// TIA Portal project "Robin_automation" (V16)
// Vorlageprojekt für das Buch mit Zielsystem S7-1200

(* hardware
DEVICE "S7-1200-Station_1"  S7-1200 Station
   slot 0: "Baugruppenträger_0"  Rack  V1.0
   slot 1: "PLC_1"  CPU 1211C DC/DC/DC  6ES7 211-1AE40-0XB0  V4.1
*)

// ===== PLC "PLC_1"  CPU 1211C DC/DC/DC =====

VAR_GLOBAL   // PLC tag table "Standard-Variablentabelle"
   "Start Button 1" AT %I0.0 : Bool;
   "Stop Button 1" AT %I0.1 : Bool;
   "Emergency Stop 1" AT %I0.2 : Bool;
   "Roller Conveyor (2m) 2" AT %Q0.0 : Bool;
   "Belt Conveyor (4m) 3" AT %Q0.1 : Bool;
   "Diffuse Sensor 1" AT %I0.3 : Bool;
   "Loadong Conveyor 1" AT %Q0.2 : Bool;
   "Diffuse Sensor 4" AT %I0.4 : Bool;
   "Diffuse Sensor 2" AT %I0.5 : Bool;
   "Chain Transfer 3 (+)" AT %Q0.4 : Bool;
   "Chain Transfer 3 (Right)" AT %Q0.5 : Bool;
   "Chain Transfer 3 (Left)" AT %Q0.6 : Bool;
   "Chain Transfer 1 (Left)" AT %Q0.7 : Bool;
   "Chain Transfer 1 (+)" AT %Q1.0 : Bool;
   "Chain Transfer 2 (Right)" AT %Q1.1 : Bool;
   "Chain Transfer 2 (+)" AT %Q1.2 : Bool;
   "Belt Conveyor (4m) 2" AT %Q1.3 : Bool;
   "Belt Conveyor (4m) 1" AT %Q1.4 : Bool;
   "Diffuse Sensor 6" AT %I0.6 : Bool;
   "Diffuse Sensor 3" AT %I0.7 : Bool;
   "Diffuse Sensor 7" AT %I1.0 : Bool;
   "Diffuse Sensor 8" AT %I1.1 : Bool;
   "Tag_1" AT %M0.0 : Bool;
   "Tag_2" AT %M0.1 : Bool;
   "Stack Light 1 (Green)" AT %Q1.7 : Bool;
   "Stack Light 1 (Yellow)" AT %Q1.6 : Bool;
   "Tag_3" AT %M0.3 : Bool;
   "Barkod Bitti" AT %I1.2 : Bool;
   "Loading Conveyor 2" AT %Q1.5 : Bool;
   "Tag_4" AT %M0.5 : Bool;
   "Tag_5" AT %M0.4 : Bool;
   "Tag_6" AT %M1.0 : Bool;
   "Tag_7" AT %M2.0 : Bool;
   "Diffuse Sensor 5" AT %I1.3 : Bool;
   "Tag_8" AT %M2.1 : Bool;
   "Tag_9" AT %M3.0 : Bool;
   "Start Button 3" AT %I1.4 : Bool;
   "Tag_10" AT %M3.1 : Bool;
   "Tag_11" AT %M1.1 : Bool;
   "Tag_12" AT %M1.2 : Bool;
   "Tag_13" AT %M1.3 : Bool;
   "Tag_14" AT %M0.2 : Bool;
   "Tag_15" AT %M1.4 : Bool;
   "Tag_16" AT %M1.5 : Bool;
   "Tag_17" AT %M1.6 : Bool;
   "Tag_18" AT %M1.7 : Bool;
   "Tag_19" AT %M0.6 : Bool;
   "Sağ boş  Sol dolu ise AÇIK" AT %M0.7 : Bool;
   "Tag_20" AT %M2.2 : Bool;
   "Tag_21" AT %M2.3 : Bool;
   "Tag_22" AT %M2.5 : Bool;
   "Tag_23" AT %M2.6 : Bool;
   "Tag_24" AT %M2.7 : Bool;
END_VAR

TYPE "User_data_type_1"
   STRUCT
      "Start Button" : Bool;
   END_STRUCT;
END_TYPE

FUNCTION "MHJ-PLC-Lab-Function-S71200" : Void   // FC9000, SCL
{ S7_Optimized_Access := 'TRUE' }
VERSION : 0.1
   VAR_TEMP
      rdTimeReturn : Int;
      outputTime : DTL;
      SyncVal : Byte;
      forVal : Int;
      forVal_2 : Int;
      Value : Byte;
   END_VAR
   VAR CONSTANT
      CompVal : Byte := 16#34;
      Value_01 : Byte := 16#11;
      Value_01_DW : DWord := 16#A165_D992;
      Value_02_DW : DWord := 16#58BE_4401;
   END_VAR
BEGIN

   #Value:=PEEK(area := 16#82,
        dbNumber := 0,
        byteOffset := 511);
   #Value := #Value + 1;

   POKE(area := 16#82,
        dbNumber := 0,
        byteOffset := 511,
        value := #Value);

   POKE(area:=16#81,
        dbNumber:=0,
        byteOffset:=1016,
        value:=#Value_01_DW);
   POKE(area := 16#81,
        dbNumber := 0,
        byteOffset := 1020,
        value := #Value_02_DW);

   POKE(area := 16#81,
        dbNumber := 0,
        byteOffset := 511,
        value := B#16#00);

   FOR #forVal := 0 TO 120 DO
       FOR #forVal_2:=0 TO 10 DO
           #rdTimeReturn:=RD_SYS_T(#outputTime);
           #rdTimeReturn := WR_SYS_T(#outputTime);
           #rdTimeReturn := RD_SYS_T(#outputTime);
           #rdTimeReturn := WR_SYS_T(#outputTime);
       END_FOR;
       #SyncVal:= PEEK(area := 16#81,
                      dbNumber := 0,
                      byteOffset := 511);
       IF #SyncVal = #CompVal THEN
          GOTO M_1;
       END_IF;
   END_FOR;
   RETURN;

   M_1:
   POKE(area := 16#81,
        dbNumber := 0,
        byteOffset := 511,
        value := B#16#0);
END_FUNCTION

// folder: System blocks/Program resources

ORGANIZATION_BLOCK "Main"   // OB1, LAD, ProgramCycle
TITLE = "Main Program Sweep (Cycle)"
{ S7_Optimized_Access := 'TRUE' }
VERSION : 0.1
   VAR_INPUT
      Initial_Call : Bool;   // Initial call of this OB
      Remanence : Bool;   // =True, if remanent data are available
   END_VAR
   VAR_TEMP   // added for the SCL form of the ladder/FBD networks
      _w1 : Bool;
      _w2 : Bool;
   END_VAR
BEGIN

REGION Network 1: Konnektierungsbaustein für PLC-Lab
   // Im Netzwerk 1 wird der Konnektierungsbaustein für PLC-Lab aufgerufen.
   // Dieser Aufruf darf nicht entfernt werden!
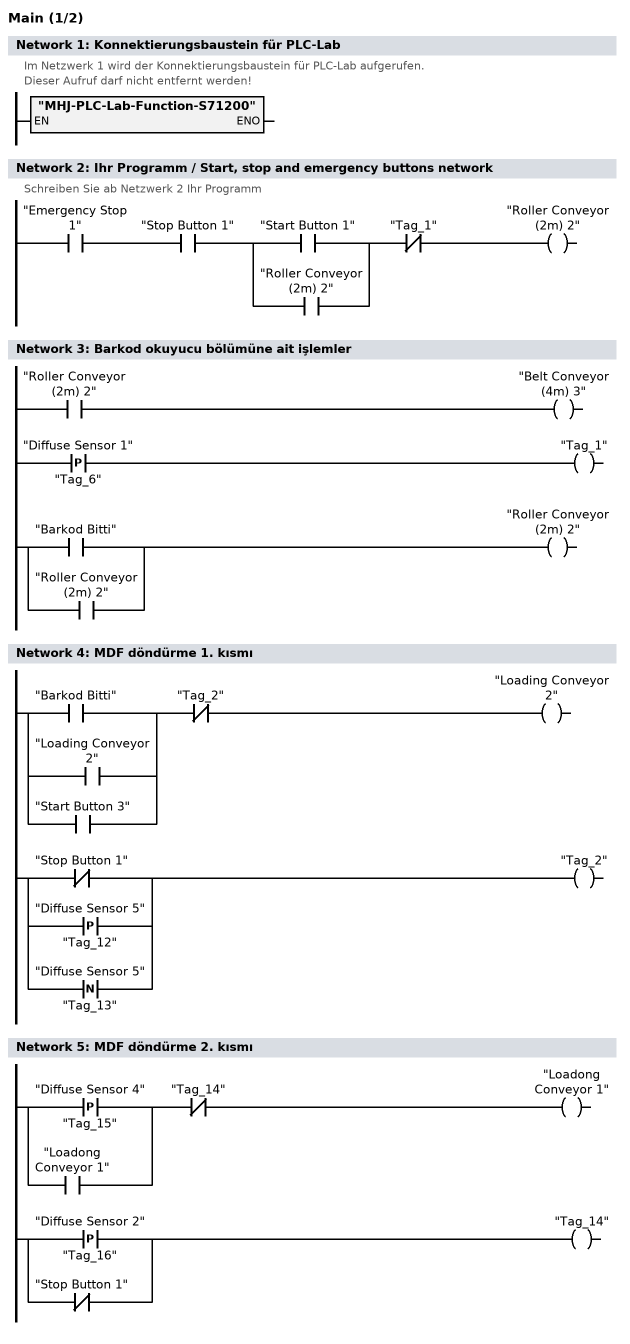
   RUNG wire#powerrail
      "MHJ-PLC-Lab-Function-S71200"()
   END_RUNG
   // the same network as SCL:
   "MHJ-PLC-Lab-Function-S71200"();
END_REGION

REGION Network 2: Ihr Programm / Start, stop and emergency buttons network
   // Schreiben Sie ab Netzwerk 2 Ihr Programm
   RUNG wire#powerrail
      Contact( "Emergency Stop 1" )
      Contact( "Stop Button 1" )
      wire#w1
      Contact( "Start Button 1" )
      wire#w2
      I_Contact( "Tag_1" )
      Coil( "Roller Conveyor (2m) 2" )
   END_RUNG
   RUNG wire#w1
      Contact( "Roller Conveyor (2m) 2" )
   END_RUNG wire#w2
   // the same network as SCL:
   "Roller Conveyor (2m) 2" := "Emergency Stop 1" AND "Stop Button 1" AND ("Start Button 1" OR "Roller Conveyor (2m) 2") AND NOT "Tag_1";
END_REGION

REGION Network 3: Barkod okuyucu bölümüne ait işlemler
   RUNG wire#powerrail
      Contact( "Roller Conveyor (2m) 2" )
      Coil( "Belt Conveyor (4m) 3" )
   END_RUNG
   RUNG wire#powerrail
      P_Contact(operand := "Diffuse Sensor 1", bit := "Tag_6")
      Coil( "Tag_1" )
   END_RUNG
   RUNG wire#powerrail
      Contact( "Barkod Bitti" )
      wire#w1
      Coil( "Roller Conveyor (2m) 2" )
   END_RUNG
   RUNG wire#powerrail
      Contact( "Roller Conveyor (2m) 2" )
   END_RUNG wire#w1
   // the same network as SCL:
   "Belt Conveyor (4m) 3" := "Roller Conveyor (2m) 2";
   #_w1 := "Diffuse Sensor 1" AND NOT "Tag_6";   // rising edge of "Diffuse Sensor 1"
   "Tag_6" := "Diffuse Sensor 1";
   "Tag_1" := #_w1;
   "Roller Conveyor (2m) 2" := "Barkod Bitti" OR "Roller Conveyor (2m) 2";
END_REGION

REGION Network 4: MDF döndürme 1. kısmı
   RUNG wire#powerrail
      Contact( "Barkod Bitti" )
      wire#w1
      I_Contact( "Tag_2" )
      Coil( "Loading Conveyor 2" )
   END_RUNG
   RUNG wire#powerrail
      Contact( "Loading Conveyor 2" )
   END_RUNG wire#w1
   RUNG wire#powerrail
      Contact( "Start Button 3" )
   END_RUNG wire#w1
   RUNG wire#powerrail
      I_Contact( "Stop Button 1" )
      wire#w2
      Coil( "Tag_2" )
   END_RUNG
   RUNG wire#powerrail
      P_Contact(operand := "Diffuse Sensor 5", bit := "Tag_12")
   END_RUNG wire#w2
   RUNG wire#powerrail
      N_Contact(operand := "Diffuse Sensor 5", bit := "Tag_13")
   END_RUNG wire#w2
   // the same network as SCL:
   "Loading Conveyor 2" := ("Barkod Bitti" OR "Loading Conveyor 2" OR "Start Button 3") AND NOT "Tag_2";
   #_w1 := "Diffuse Sensor 5" AND NOT "Tag_12";   // rising edge of "Diffuse Sensor 5"
   "Tag_12" := "Diffuse Sensor 5";
   #_w2 := NOT "Diffuse Sensor 5" AND "Tag_13";   // falling edge of "Diffuse Sensor 5"
   "Tag_13" := "Diffuse Sensor 5";
   "Tag_2" := NOT "Stop Button 1" OR #_w1 OR #_w2;
END_REGION

REGION Network 5: MDF döndürme 2. kısmı
   RUNG wire#powerrail
      P_Contact(operand := "Diffuse Sensor 4", bit := "Tag_15")
      wire#w1
      I_Contact( "Tag_14" )
      Coil( "Loadong Conveyor 1" )
   END_RUNG
   RUNG wire#powerrail
      Contact( "Loadong Conveyor 1" )
   END_RUNG wire#w1
   RUNG wire#powerrail
      P_Contact(operand := "Diffuse Sensor 2", bit := "Tag_16")
      wire#w2
      Coil( "Tag_14" )
   END_RUNG
   RUNG wire#powerrail
      I_Contact( "Stop Button 1" )
   END_RUNG wire#w2
   // the same network as SCL:
   #_w1 := "Diffuse Sensor 4" AND NOT "Tag_15";   // rising edge of "Diffuse Sensor 4"
   "Tag_15" := "Diffuse Sensor 4";
   "Loadong Conveyor 1" := (#_w1 OR "Loadong Conveyor 1") AND NOT "Tag_14";
   #_w2 := "Diffuse Sensor 2" AND NOT "Tag_16";   // rising edge of "Diffuse Sensor 2"
   "Tag_16" := "Diffuse Sensor 2";
   "Tag_14" := #_w2 OR NOT "Stop Button 1";
END_REGION

REGION Network 6: Orta kısım
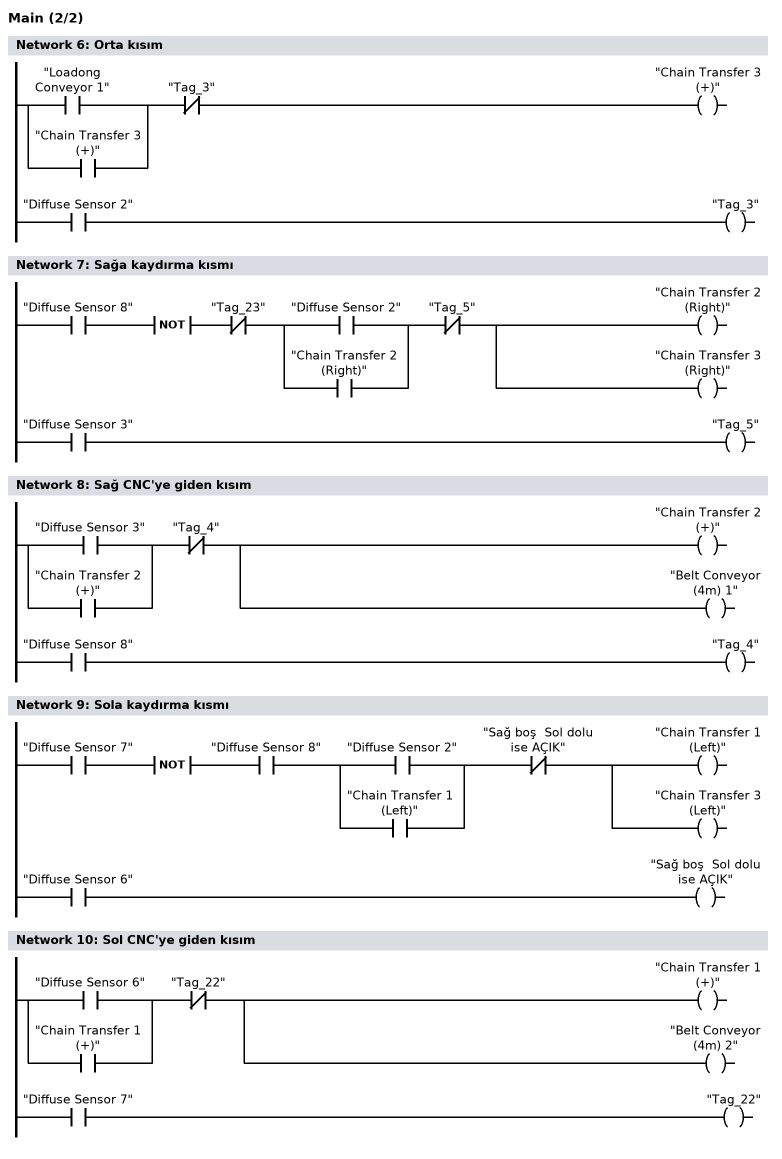
   RUNG wire#powerrail
      Contact( "Loadong Conveyor 1" )
      wire#w1
      I_Contact( "Tag_3" )
      Coil( "Chain Transfer 3 (+)" )
   END_RUNG
   RUNG wire#powerrail
      Contact( "Chain Transfer 3 (+)" )
   END_RUNG wire#w1
   RUNG wire#powerrail
      Contact( "Diffuse Sensor 2" )
      Coil( "Tag_3" )
   END_RUNG
   // the same network as SCL:
   "Chain Transfer 3 (+)" := ("Loadong Conveyor 1" OR "Chain Transfer 3 (+)") AND NOT "Tag_3";
   "Tag_3" := "Diffuse Sensor 2";
END_REGION

REGION Network 7: Sağa kaydırma kısmı
   RUNG wire#powerrail
      Contact( "Diffuse Sensor 8" )
      Not()
      I_Contact( "Tag_23" )
      wire#w1
      Contact( "Diffuse Sensor 2" )
      wire#w2
      I_Contact( "Tag_5" )
      wire#w3
      Coil( "Chain Transfer 2 (Right)" )
   END_RUNG
   RUNG wire#w1
      Contact( "Chain Transfer 2 (Right)" )
   END_RUNG wire#w2
   RUNG wire#w3
      Coil( "Chain Transfer 3 (Right)" )
   END_RUNG
   RUNG wire#powerrail
      Contact( "Diffuse Sensor 3" )
      Coil( "Tag_5" )
   END_RUNG
   // the same network as SCL:
   "Chain Transfer 2 (Right)" := NOT "Diffuse Sensor 8" AND NOT "Tag_23" AND ("Diffuse Sensor 2" OR "Chain Transfer 2 (Right)") AND NOT "Tag_5";
   "Chain Transfer 3 (Right)" := "Chain Transfer 2 (Right)";
   "Tag_5" := "Diffuse Sensor 3";
END_REGION

REGION Network 8: Sağ CNC'ye giden kısım
   RUNG wire#powerrail
      Contact( "Diffuse Sensor 3" )
      wire#w1
      I_Contact( "Tag_4" )
      wire#w2
      Coil( "Chain Transfer 2 (+)" )
   END_RUNG
   RUNG wire#powerrail
      Contact( "Chain Transfer 2 (+)" )
   END_RUNG wire#w1
   RUNG wire#w2
      Coil( "Belt Conveyor (4m) 1" )
   END_RUNG
   RUNG wire#powerrail
      Contact( "Diffuse Sensor 8" )
      Coil( "Tag_4" )
   END_RUNG
   // the same network as SCL:
   "Chain Transfer 2 (+)" := ("Diffuse Sensor 3" OR "Chain Transfer 2 (+)") AND NOT "Tag_4";
   "Belt Conveyor (4m) 1" := "Chain Transfer 2 (+)";
   "Tag_4" := "Diffuse Sensor 8";
END_REGION

REGION Network 9: Sola kaydırma kısmı
   RUNG wire#powerrail
      Contact( "Diffuse Sensor 7" )
      Not()
      Contact( "Diffuse Sensor 8" )
      wire#w1
      Contact( "Diffuse Sensor 2" )
      wire#w2
      I_Contact( "Sağ boş  Sol dolu ise AÇIK" )
      wire#w3
      Coil( "Chain Transfer 1 (Left)" )
   END_RUNG
   RUNG wire#w1
      Contact( "Chain Transfer 1 (Left)" )
   END_RUNG wire#w2
   RUNG wire#w3
      Coil( "Chain Transfer 3 (Left)" )
   END_RUNG
   RUNG wire#powerrail
      Contact( "Diffuse Sensor 6" )
      Coil( "Sağ boş  Sol dolu ise AÇIK" )
   END_RUNG
   // the same network as SCL:
   "Chain Transfer 1 (Left)" := NOT "Diffuse Sensor 7" AND "Diffuse Sensor 8" AND ("Diffuse Sensor 2" OR "Chain Transfer 1 (Left)") AND NOT "Sağ boş  Sol dolu ise AÇIK";
   "Chain Transfer 3 (Left)" := "Chain Transfer 1 (Left)";
   "Sağ boş  Sol dolu ise AÇIK" := "Diffuse Sensor 6";
END_REGION

REGION Network 10: Sol CNC'ye giden kısım
   RUNG wire#powerrail
      Contact( "Diffuse Sensor 6" )
      wire#w1
      I_Contact( "Tag_22" )
      wire#w2
      Coil( "Chain Transfer 1 (+)" )
   END_RUNG
   RUNG wire#powerrail
      Contact( "Chain Transfer 1 (+)" )
   END_RUNG wire#w1
   RUNG wire#w2
      Coil( "Belt Conveyor (4m) 2" )
   END_RUNG
   RUNG wire#powerrail
      Contact( "Diffuse Sensor 7" )
      Coil( "Tag_22" )
   END_RUNG
   // the same network as SCL:
   "Chain Transfer 1 (+)" := ("Diffuse Sensor 6" OR "Chain Transfer 1 (+)") AND NOT "Tag_22";
   "Belt Conveyor (4m) 2" := "Chain Transfer 1 (+)";
   "Tag_22" := "Diffuse Sensor 7";
END_REGION
END_ORGANIZATION_BLOCK